// This interface defines the behaviour of a timer, a type of timing source used
// to track a specific duration. The timer can be started, paused, stopped, and
// cleared. It is commonly used for timing events, delays, and other time-based
// operations. The timer tracks elapsed time and can indicate when the set 
// duration has expired.
INTERFACE I_Timer EXTENDS I_TimingSource

// Clears the timer, resetting the elapsed time.
METHOD Clear
VAR_INPUT
END_VAR
END_METHOD

// The duration for the timer. It specifies how long the timer should run before
// it expires.
// [get] Returns the set duration.
// [set] Sets the duration for the timer.
PROPERTY Duration : LTIME
GET
END_GET
SET
END_SET
END_PROPERTY

// The elapsed time since the timer was started.
// [get] Returns the elapsed time.
PROPERTY ElapsedTime  : LTIME
GET
END_GET
END_PROPERTY

// Indicates whether the timer has expired.
// [get] Returns TRUE if the timer has expired; otherwise, FALSE.
PROPERTY HasExpired : BOOL
GET
END_GET
END_PROPERTY

// Indicates whether the timer is currently paused.
// [get] Returns TRUE if the timer is paused; otherwise, FALSE.
PROPERTY HasPaused : BOOL
GET
END_GET
END_PROPERTY

// Indicates whether the timer is currently running.
// [get] Returns TRUE if the timer is running; otherwise, FALSE.
PROPERTY IsRunning  : BOOL
GET
END_GET
END_PROPERTY

// Pauses the timer, preserving the elapsed time without resetting.
METHOD Pause
VAR_INPUT
END_VAR
END_METHOD

// Starts the timer, beginning the tracking of time towards the specified duration.
METHOD Start
VAR_INPUT
END_VAR
END_METHOD

// Stops the timer, halting the tracking of time.
METHOD Stop
VAR_INPUT
END_VAR
END_METHOD

// The remaining time until the timer expires.
// [get] Returns the time remaining until expiration.
PROPERTY TimeRemaining : LTIME
GET
END_GET
END_PROPERTY

END_INTERFACE

(* stored: Version 1.1.0.1
   Itf I_Timer: Id {9f15de56-b770-4791-88f8-757da808d4d1}
   Method Clear: Id {fbde5924-6508-4072-84d4-3ac33b125a5c}
   Property Duration: Id {cd088390-8b66-43ef-8045-c7e3bf5c9701}
   Get Get: Id {4b342c9b-964b-4324-acc0-5b8e596292e2}
   Set Set: Id {c0d7d71b-ee01-40fa-89e1-191f7c5d12be}
   Property ElapsedTime: Id {1fbfb67b-8cc7-45f9-825b-708932e30068}
   Get Get: Id {b4ffe30e-7377-4327-8142-55cacc649397}
   Property HasExpired: Id {9f743a48-2302-45ca-a2c2-a132cfcef96b}
   Get Get: Id {babdbfeb-d5d6-4502-b862-2e5bf76f011f}
   Property HasPaused: Id {8d7afcd9-7c45-49f3-8d41-c28892d21654}
   Get Get: Id {b14d3f7a-9dbc-47db-8565-c1f35ad4c874}
   Property IsRunning: Id {5a4a3611-16fb-41fc-8b0f-72af0a004b68}
   Get Get: Id {7183ac11-ec3b-4529-98d0-7bf2b16d602e}
   Method Pause: Id {d21a3ad5-3bae-03fe-323c-88951657accd}
   Method Start: Id {eeabeabc-df7e-4218-8966-f6444ad9be0a}
   Method Stop: Id {96644411-9fc8-4775-872e-6081ca03f88e}
   Property TimeRemaining: Id {3ce45e66-5e6b-4f1c-ab26-bc71712154fa}
   Get Get: Id {c17b6151-ded3-4707-b79b-99d76272e200} *)
